# EPICS autosave request: apps/iocBoot/iocmyaData/harpScanDataAll.req
file harpScanData.req P=HB_BEAM:SCAN:,R=2c21:
file harpScanData.req P=HB_BEAM:SCAN:,R=tagger:
file harpScanData.req P=HB_BEAM:SCAN:,R=2H02A:
